FUNCTION_BLOCK VentilationControl
VAR_INPUT
	EN: BOOL;
	StopFans: BOOL;
END_VAR
VAR_OUTPUT
	ENO: BOOL;
END_VAR
VAR
END_VAR
VAR PERSISTENT
END_VAR

ENO := EN AND NOT StopFans;

END_FUNCTION_BLOCK

(* stored: Version 1.1.0.1, ProductVersion 3.1.4024.6
   POU VentilationControl: Id {d0f91fb4-6566-4ba9-86f0-d920b5d00d5c}, SpecialFunc None *)
